{attribute addProperty BoxType "EJ4004-0000-0020"}
{attribute addProperty Id "AO_Outputs_ChannelAT %Q*ARRAY[0..3] OF AO_Outputs_Channel_F57FA4F96480WcStateAT %I*WcState_64F6A8C6810InfoDataAT %I*InfoData_BC63D37F80100"}
{attribute addProperty CRC "645842055"}
{attribute addProperty SizeInBites "152"}
{attribute addProperty SizeInBytes "19"}
TYPE EJ4004_253CF8AE :
STRUCT
	{attribute addProperty Name "AO_Outputs_Channel"}
	AO_Outputs_Channel : ARRAY[0..3] OF AO_Outputs_Channel_F57FA4F9;
	{attribute addProperty Name "WcState"}
	WcState : WcState_64F6A8C6;
	{attribute addProperty Name "InfoData"}
	InfoData : InfoData_BC63D37F;
END_STRUCT
END_TYPE

(* stored: Version 1.2.0.0, ProductVersion 3.1.4024.9
   DUT EJ4004_253CF8AE: Id {1f321145-fef5-4414-9d90-78b8a311f8f4} *)
